// TIA Portal V21 export
DATA_BLOCK "DigitalOutput_DB"   // DB5
// stored: InstanceOfName DigitalOutput, InstanceOfType FB
"DigitalOutput"
   // VAR_INPUT
   //    Cmd { ExternalVisible := 'False'} : Bool;
   //    SimulationOn { ExternalVisible := 'False'} : Bool;
   //    MotorFeedbackInputSelection { ExternalVisible := 'False'} : Bool;
   //    MotorFeedbackInput { ExternalVisible := 'False'} : Bool;
   //    WaterSensorSelection { ExternalVisible := 'False'} : Bool;
   //    WaterSensorInput { ExternalVisible := 'False'} : Bool;
   //    AlwaysTrue : Bool;
   //    AlwaysFalse : Bool;
   //    OpenClose : Bool;
   //    Spare_3 : Bool;
   //    ValveFeedbackInputSelection { ExternalVisible := 'False'} : Bool;
   //    ValveFeedbackInput { ExternalVisible := 'False'} : Bool;
   //    Interlock : Bool;
   //    FBCheckDelay { ExternalVisible := 'False'} : Int;
   //    WSCheckDelay { ExternalVisible := 'False'} : Int;
   //    secs { ExternalVisible := 'False'} : Bool;
   //    AlarmAck { ExternalVisible := 'False'} : Bool;
   //    ModeSel : Bool;
   //    Fault : Bool;
   //    Reset : Bool;
   //    spare : Bool;
   //    spare_1 : Bool;
   //    spare_2 : Bool;
   // END_VAR
   // VAR_OUTPUT
   //    Output { ExternalVisible := 'False'} : Bool;
   //    FeedBackTripAlarm : Bool;
   //    NoWaterFlowAlarm : Bool;
   //    LineColour : DInt;
   //    ValveColour : DInt;
   //    Mode : DInt;
   //    Status : DInt;
   // END_VAR
   // VAR_IN_OUT
   //    OpFbTrip { ExternalVisible := 'False'} : Bool;
   //    OpWaterSensorTrip { ExternalVisible := 'False'} : Bool;
   //    FBCheckActualTime { ExternalVisible := 'False'} : Int;
   //    WSCheckActualTime { ExternalVisible := 'False'} : Int;
   // END_VAR
   // VAR
   //    ResetBtn { S7_SetPoint := 'True'} : TON_TIME;
   // END_VAR
BEGIN
END_DATA_BLOCK
